Fanuc KAREL source: kx00021.KL

-- PROVISIONAL review KL for V770-1; original PC SHA256 0831e62d484dee0d38c1e164d828c36052d077b5b08cf899d0d825cc44298bef
-- Incomplete behavior may be omitted. Consult companion uncertainty JSON. Do not deploy.
PROGRAM KX00021
%NOLOCKGROUP
BEGIN
  -- UNRESOLVED_PC offsets 5-25; opcodes 2E,22,9D,33,2E,33,35
  -- UNRESOLVED_PC offsets 30-51; opcodes 22,9D,33,2E,33,34,23
  -- UNRESOLVED_PC offsets 56-60; opcodes 7F
END KX00021
